FUNCTION_BLOCK SC_PrePalletizer EXTENDS FB_Chain
VAR_INPUT
	bPalletizerRequest : BOOL;
	bExecute : BOOL;
END_VAR
VAR_OUTPUT
	bSentToPalletizer : BOOL;
	bPalletAvailable : BOOL;
END_VAR
VAR
	fbRollConvEntrance : RollerConveyor;
	fbRollConvPrePallet : RollerConveyor;
	fbPalletAvailable : Sensor;
END_VAR

SUPER^();
fbPalletAvailable();
bPalletAvailable := fbPalletAvailable.bSignal;

METHOD PROTECTED   Busy : BOOL
VAR_INPUT
END_VAR
fbStepWorkerBusy();
CASE fbStepWorkerBusy.uiStep OF
	
	0: 
		fbRollConvEntrance.On();
		fbRollConvPrePallet.On();
		IF NOT bPalletAvailable
		THEN
			bSentToPalletizer := TRUE;
			fbStepWorkerBusy.mNextStep(10);
		END_IF

	10:
		IF NOT bPalletizerRequest
		THEN
		
			bSentToPalletizer := FALSE;
			fbRollConvPrePallet.Off();
			fbStepWorkerBusy.mNextStep(0);
			
			Done();
			
		ELSIF bPalletAvailable
		THEN
			fbRollConvEntrance.Off();
		END_IF
		
END_CASE
END_METHOD

METHOD PROTECTED  Error : BOOL
VAR_INPUT
END_VAR
END_METHOD

METHOD PROTECTED  Idle : BOOL
VAR_INPUT
END_VAR
END_METHOD

METHOD PROTECTED  Init : BOOL
VAR_INPUT
END_VAR
Start();
END_METHOD

METHOD PROTECTED  Prepare : BOOL
VAR_INPUT
END_VAR
END_METHOD

METHOD PROTECTED  Ready : BOOL
VAR_INPUT
END_VAR

fbStepWorkerReady();
CASE fbStepWorkerReady.uiStep OF
	
	0:
		IF bExecute
		THEN
			fbStepWorkerReady.mNextStep(5);
		END_IF
		
	5: 
		IF NOT bPalletAvailable
		THEN
			fbRollConvEntrance.On();
		ELSIF bPalletAvailable
		THEN
			fbRollConvEntrance.Off();
			fbStepWorkerReady.mNextStep(10);
		END_IF
		
	10:
		IF bPalletizerRequest
		THEN
			fbStepWorkerReady.mNextStep(0);
			Execute();
		END_IF
		
END_CASE
END_METHOD

METHOD PROTECTED  Waiting : BOOL
VAR_INPUT
END_VAR
END_METHOD

END_FUNCTION_BLOCK

(* stored: Version 1.1.0.1, ProductVersion 3.1.4024.2
   POU SC_PrePalletizer: Id {4d68b7a9-380f-4680-8c23-9b189695cad0}, SpecialFunc None
   Method Busy: Id {d820917f-4e25-46f9-9d52-32a81aa4f13f}
   Method Error: Id {46485dc9-f0d7-4867-b360-d540fed53e71}
   Method Idle: Id {6c9d5d66-bd5f-4610-99f9-63f453dbc70c}
   Method Init: Id {09f332ae-57ff-4d70-8e40-ebbc7ec6148e}
   Method Prepare: Id {fb8b9c49-3513-4272-b7c4-bbd7656237ef}
   Method Ready: Id {f44ab75c-fea3-477e-acab-1329dc0b9d52}
   Method Waiting: Id {77554b89-ed18-4d33-9356-fca189e07525} *)
